// TIA Portal V19 export
TYPE "UDT_STATUS_MTRDIR"
   STRUCT
      running : Bool;
      inFault : Bool;
      justStarted : Bool;
      justStopped : Bool;
      justHadFault { ExternalAccessible := 'False'; ExternalVisible := 'False'; ExternalWritable := 'False'} : Bool;
      justLostFault { ExternalAccessible := 'False'; ExternalVisible := 'False'; ExternalWritable := 'False'} : Bool;
      enabled { ExternalAccessible := 'False'; ExternalVisible := 'False'; ExternalWritable := 'False'} : Bool;
      old : Struct
         running : Bool;
         fault : Bool;
      END_STRUCT;
   END_STRUCT;
END_TYPE
